INTERFACE ITF_Base

METHOD Disable : BOOL
VAR_INPUT
END_VAR
END_METHOD

METHOD Enable : BOOL
VAR_INPUT
END_VAR
END_METHOD

PROPERTY EnableNegativeDirection : bool
GET
END_GET
SET
END_SET
END_PROPERTY

PROPERTY Override : lreal
GET
END_GET
SET
END_SET
END_PROPERTY

METHOD Reset : BOOL
VAR_INPUT
END_VAR
END_METHOD

END_INTERFACE

(* stored: Version 1.1.0.1, ProductVersion 3.1.4024.3
   Itf ITF_Base: Id {7c0b5f35-6961-401c-a129-c286a521a6d4}
   Method Disable: Id {841ea02a-a785-4841-af47-9ea4c09af8f2}
   Method Enable: Id {4f565508-8f93-4c28-901f-5eaf0c6c6987}
   Property EnableNegativeDirection: Id {79b8ffa5-86f4-46fa-8e6d-3ee24842e46f}
   Get Get: Id {a6662a0e-841e-4315-9bf0-606c3c29810f}
   Set Set: Id {a0270660-c8a3-45a3-9d33-1cdbb5fae15c}
   Property Override: Id {279d333c-cb93-4282-b275-6bc17aa72e2b}
   Get Get: Id {07367dfe-a7a1-485e-9ced-ce128cae3c11}
   Set Set: Id {63842dd0-fbce-45b5-89a8-d3c548a80219}
   Method Reset: Id {171c9372-db41-483a-a539-db6009a86252} *)
